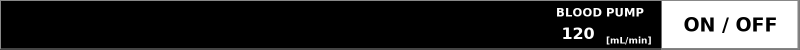
VISUALIZATION Footer  // 800x50
    Rectangle (0,0 800x50)
    Button (661,0 139x50), "ON / OFF"
    Textfield (550,0 100x25), "BLOOD PUMP"
    Textfield (528,21 100x25), "120"
    Textfield (579,28 100x25), "[mL/min]"
END_VISUALIZATION

(* stored: Version 1.1.0.1, ProductVersion 3.1.4024.12
   Visu Footer: Id {ba1b7073-6077-4d99-b632-2173f2934877} *)
